(* CODESYS project Storage.project

Project tree, tasks and I/O mapping:
  Storage : CECC-LK, Festo AG & Co. KG, order no. 574418, version 3.5.4.0
    application Application
      libraries: Util, * (System)
      task MainTask (cyclic, interval t#20ms, priority 20) calls Main
      global variables GVL_Storage
      function block FB_BitCode [SFC]: ACT
      function block FB_SeqNTransport_ST [SFC]: ACT
      function block FB_OpMode [FBD]
      program Main [FBD]
    Onboard : CECC 14I/8O, Festo AG & Co. KG, order no. 
      , version 3.4.5.5
        unmapped channels: Onboard Input, Onboard Output
      Digital Inputs
          unmapped channels: Onboard Input
      Digital Outputs
          unmapped channels: Onboard Output
    IO_Link_Master_4_Ports_ : IO-Link Master (4 Ports), Festo AG & Co. KG, order no. 
      , version 3.0.0.3
      BNI_IOL_310_000_K025 : BNI IOL-310-000-K025, Balluff GmbH, version V1.2
          settings:  = 0; ProcessDataID = V_PdT; ProcessDataInLength = 16; ProcessDataOutLength = 16; ProcessDataDescription.bitOffset = 8; ProcessDataDescription.bitLength = 1; ProcessDataDescription.userType = 0; ProcessDataDescription.ChannelType = 1; ProcessDataDescription.bitOffset = 9; ProcessDataDescription.bitLength = 1; ProcessDataDescription.userType = 0; ProcessDataDescription.ChannelType = 1; ProcessDataDescription.bitOffset = 10; ProcessDataDescription.bitLength = 1; ProcessDataDescription.userType = 0; ProcessDataDescription.ChannelType = 1; ProcessDataDescription.bitOffset = 11; ProcessDataDescription.bitLength = 1; ProcessDataDescription.userType = 0; ProcessDataDescription.ChannelType = 1; ProcessDataDescription.bitOffset = 12; ProcessDataDescription.bitLength = 1; ProcessDataDescription.userType = 0; ProcessDataDescription.ChannelType = 1; ProcessDataDescription.bitOffset = 13; ProcessDataDescription.bitLength = 1; ProcessDataDescription.userType = 0; ProcessDataDescription.ChannelType = 1; ProcessDataDescription.bitOffset = 14; ProcessDataDescription.bitLength = 1; ProcessDataDescription.userType = 0; ProcessDataDescription.ChannelType = 1; ProcessDataDescription.bitOffset = 15; ProcessDataDescription.bitLength = 1; ProcessDataDescription.userType = 0; ProcessDataDescription.ChannelType = 1; ProcessDataDescription.bitOffset = 0; ProcessDataDescription.bitLength = 1; ProcessDataDescription.userType = 0; ProcessDataDescription.ChannelType = 1;
            ProcessDataDescription.bitOffset = 1; ProcessDataDescription.bitLength = 1; ProcessDataDescription.userType = 0; ProcessDataDescription.ChannelType = 1; ProcessDataDescription.bitOffset = 2; ProcessDataDescription.bitLength = 1; ProcessDataDescription.userType = 0; ProcessDataDescription.ChannelType = 1; ProcessDataDescription.bitOffset = 3; ProcessDataDescription.bitLength = 1; ProcessDataDescription.userType = 0; ProcessDataDescription.ChannelType = 1; ProcessDataDescription.bitOffset = 4; ProcessDataDescription.bitLength = 1; ProcessDataDescription.userType = 0; ProcessDataDescription.ChannelType = 1; ProcessDataDescription.bitOffset = 5; ProcessDataDescription.bitLength = 1; ProcessDataDescription.userType = 0; ProcessDataDescription.ChannelType = 1; ProcessDataDescription.bitOffset = 6; ProcessDataDescription.bitLength = 1; ProcessDataDescription.userType = 0; ProcessDataDescription.ChannelType = 1; ProcessDataDescription.bitOffset = 7; ProcessDataDescription.bitLength = 1; ProcessDataDescription.userType = 0; ProcessDataDescription.ChannelType = 1; ProcessDataDescription.bitOffset = 8; ProcessDataDescription.bitLength = 1; ProcessDataDescription.userType = 0; ProcessDataDescription.ChannelType = 2; ProcessDataDescription.bitOffset = 9; ProcessDataDescription.bitLength = 1; ProcessDataDescription.userType = 0; ProcessDataDescription.ChannelType = 2; ProcessDataDescription.bitOffset = 10; ProcessDataDescription.bitLength = 1; ProcessDataDescription.userType = 0; ProcessDataDescription.ChannelType = 2;
            ProcessDataDescription.bitOffset = 11; ProcessDataDescription.bitLength = 1; ProcessDataDescription.userType = 0; ProcessDataDescription.ChannelType = 2; ProcessDataDescription.bitOffset = 12; ProcessDataDescription.bitLength = 1; ProcessDataDescription.userType = 0; ProcessDataDescription.ChannelType = 2; ProcessDataDescription.bitOffset = 13; ProcessDataDescription.bitLength = 1; ProcessDataDescription.userType = 0; ProcessDataDescription.ChannelType = 2; ProcessDataDescription.bitOffset = 14; ProcessDataDescription.bitLength = 1; ProcessDataDescription.userType = 0; ProcessDataDescription.ChannelType = 2; ProcessDataDescription.bitOffset = 15; ProcessDataDescription.bitLength = 1; ProcessDataDescription.userType = 0; ProcessDataDescription.ChannelType = 2; ProcessDataDescription.bitOffset = 0; ProcessDataDescription.bitLength = 1; ProcessDataDescription.userType = 0; ProcessDataDescription.ChannelType = 2; ProcessDataDescription.bitOffset = 1; ProcessDataDescription.bitLength = 1; ProcessDataDescription.userType = 0; ProcessDataDescription.ChannelType = 2; ProcessDataDescription.bitOffset = 2; ProcessDataDescription.bitLength = 1; ProcessDataDescription.userType = 0; ProcessDataDescription.ChannelType = 2; ProcessDataDescription.bitOffset = 3; ProcessDataDescription.bitLength = 1; ProcessDataDescription.userType = 0; ProcessDataDescription.ChannelType = 2; ProcessDataDescription.bitOffset = 4; ProcessDataDescription.bitLength = 1; ProcessDataDescription.userType = 0; ProcessDataDescription.ChannelType = 2;
            ProcessDataDescription.bitOffset = 5; ProcessDataDescription.bitLength = 1; ProcessDataDescription.userType = 0; ProcessDataDescription.ChannelType = 2; ProcessDataDescription.bitOffset = 6; ProcessDataDescription.bitLength = 1; ProcessDataDescription.userType = 0; ProcessDataDescription.ChannelType = 2; ProcessDataDescription.bitOffset = 7; ProcessDataDescription.bitLength = 1; ProcessDataDescription.userType = 0; ProcessDataDescription.ChannelType = 2
          unmapped channels: Switchstate Pin 1 (Bit0.0), Switchstate Pin 2 (Bit0.1), Switchstate Pin 3 (Bit0.2), Switchstate Pin 4 (Bit0.3), Switchstate Pin 5 (Bit0.4), Switchstate Pin 6 (Bit0.5), Switchstate Pin 7 (Bit0.6), Switchstate Pin 8 (Bit0.7), Switchstate Pin 9 (Bit1.0), Switchstate Pin 10 (Bit1.1), Switchstate Pin 11 (Bit1.2), Switchstate Pin 12 (Bit1.3), Switchstate Pin 13 (Bit1.4), Switchstate Pin 14 (Bit1.5), Switchstate Pin 15 (Bit1.6), Switchstate Pin 16 (Bit1.7), Switchstate Pin 1 (Bit0.0), Switchstate Pin 2 (Bit0.1), Switchstate Pin 3 (Bit0.2), Switchstate Pin 4 (Bit0.3), Switchstate Pin 5 (Bit0.4), Switchstate Pin 6 (Bit0.5), Switchstate Pin 7 (Bit0.6), Switchstate Pin 8 (Bit0.7), Switchstate Pin 9 (Bit1.0), Switchstate Pin 10 (Bit1.1), Switchstate Pin 11 (Bit1.2), Switchstate Pin 12 (Bit1.3), Switchstate Pin 13 (Bit1.4), Switchstate Pin 14 (Bit1.5), Switchstate Pin 15 (Bit1.6), Switchstate Pin 16 (Bit1.7)
      <Leer>
      <Leer>
      <Leer>
  libraries: Standard, * (System); Util, * (System)
  global variables ToDo
*)

// ToDo
VAR_GLOBAL
END_VAR

// Storage/Application/GVL_Storage
VAR_GLOBAL

//Input			
//Balluf IO-LINK 
xStore_ResetReady	AT	%IX2.0	:BOOL;	//
xStore_Error		AT	%IX2.1	:BOOL;	//
xStore_Busy			AT	%IX2.2	:BOOL;	//
xStore_Full			AT	%IX2.3	:BOOL;	//
xStore_WPAvailable	AT	%IX2.4	:BOOL;	//
xWPnotBlack			AT	%IX2.5	:BOOL;	//
xWPmetallic			AT	%IX2.6	:BOOL;	//
//AT	%IX2.7	:BOOL;	//
	
//CECC-LK Onboard		
SF1 	AT	%IX0.0	:BOOL;	//Taster Start / Start button
SF2 	AT	%IX0.1	:BOOL;	//Taster Stop (Öffner) / Stop Button (normally closed)
SF3 	AT	%IX0.3	:BOOL;	//Taster Richten / Reset button
SF4 	AT	%IX0.2	:BOOL;	//Schlüsselschalter Auto-Manuell / Key Switch auto-manual
XI4		AT	%IX0.4	:BOOL;	//Input from the onboard input pins 
XI5		AT	%IX0.6	:BOOL;	//
XD6 	AT	%IX0.7	:BOOL;	//Folgestation belegt / dwonstream station free			switched address with xd7 for consistency with other stations
XD7		AT	%IX0.5	:BOOL;	//Folgestation belegt / next station free			switched address with xd6 for consistency with other stations
			
//Output	
//Balluf IO-LINK 		//find out how the the xStore_BitCodeBit# is mapped with the IO
xStore_Reference	AT	%QX2.0	:BOOL;	//
xStore_ClearFault	AT	%QX2.1	:BOOL;	//
xStore_Mode			AT	%QX2.2	:BOOL;	// 0 == Store ; 1 == Unstore
xStore_BitCodeBit0	AT	%QX2.3	:BOOL;	//
xStore_BitCodeBit1	AT	%QX2.4	:BOOL;	// 
xStore_BitCodeBit2	AT	%QX2.5	:BOOL;	//
xStore_Strobe		AT	%QX2.6	:BOOL;	//
xStore_Option		AT	%QX2.7	:BOOL;	//
		
//CECC-LK Onboard	
PF1			AT	%QX0.0	:BOOL;	//Leuchtmelder Start / Start indicator light
PF2 		AT	%QX0.1	:BOOL;	//Leuchtmelder Reset / Reset indicator light
PF3 		AT	%QX0.2	:BOOL;	//Leuchte Q1 / Indicator light Q1
PF4			AT	%QX0.3	:BOOL;	//Leuchte Q2 / Indicator light Q2
XD4			AT	%QX0.4	:BOOL;	//Station frei / Station free
indLightGn	AT	%QX0.5	:BOOL;	//Ampel grün / indicator lights green
indLightYe	AT	%QX0.6	:BOOL;	//Ampel gelb / indicator lights yellow
indLightRd 	AT	%QX0.7	:BOOL;	//Apel rot / indicator lights red

// Flags for the Main prg
xStopStoring			:BOOL;
xResetModules			:BOOL;	//Alle Module resetten / Reset all Moduls
xResetReadyModule1		:BOOL;	//Module 1 ist in reset Position / Modul 1 is in reset posisition
xResetReadyModule2		:BOOL;	//Module 2 ist in reset Position / Modul 2 is in reset posisition
xResetReadyModule3		:BOOL;	//Module 3 ist in reset Position / Modul 3 is in reset posisition
xEnAutoMM				:BOOL;	//Automatikmodus aktiv / Automode activated
xDeactivateModules		:BOOL;	//
xProcessBusyMM			:BOOL;	//Station arbeitet / Station is busy
xResetReadyMM			:BOOL;	//Modul SeqTransport ist fertig / Modul SeqTransport is ready
xNextStationFreeMM		:BOOL;	//Nächste Station ist frei / Next Station is free
xReadyModSM				:BOOL;	//Modul ist fertig / Modul is ready
xStartModuleSM			:BOOL;	//Modul starten / Start modul
xInitModules			:BOOL;	//Moduel auf Inischritt setzten / Set moduls to init step
AlwaysTRUE				:BOOL:=TRUE;	//Immer true / Always true
AlwaysFALSE				:BOOL:=FALSE;	//Immer false / Always false
xErrorSignal1			:BOOL;	//Error Signal 1 / Error signal	1
xErrorSignal2			:BOOL;	//Error Signal 2 / Error signal	2
xErrorSignal3			:BOOL;	//Error Signal 3 / Error signal	3

xMKeySwitchOut			:BOOL;
xMStartOut				:BOOL;
xMI4Out					:BOOL;
xMBit0					:BOOL;
xMBit1					:BOOL;
xMBit2					:BOOL;
xMI7Out					:BOOL;
xMPF3					:BOOL;
END_VAR

// Storage/Application/Main
PROGRAM Main//the sequensce of operations 

//for the reference of the variables 
VAR
	FB_OpMode_0				: FB_OpMode; // the initialising code, and for the detection of the colour
	//xMI4Out has something to do with the rising edge from the sensors
	FB_SeqNTransport_ST_0	: FB_SeqNTransport_ST;
	//xMBits are probably for the storage location 
	FB_BitCode_0			: FB_BitCode;
END_VAR

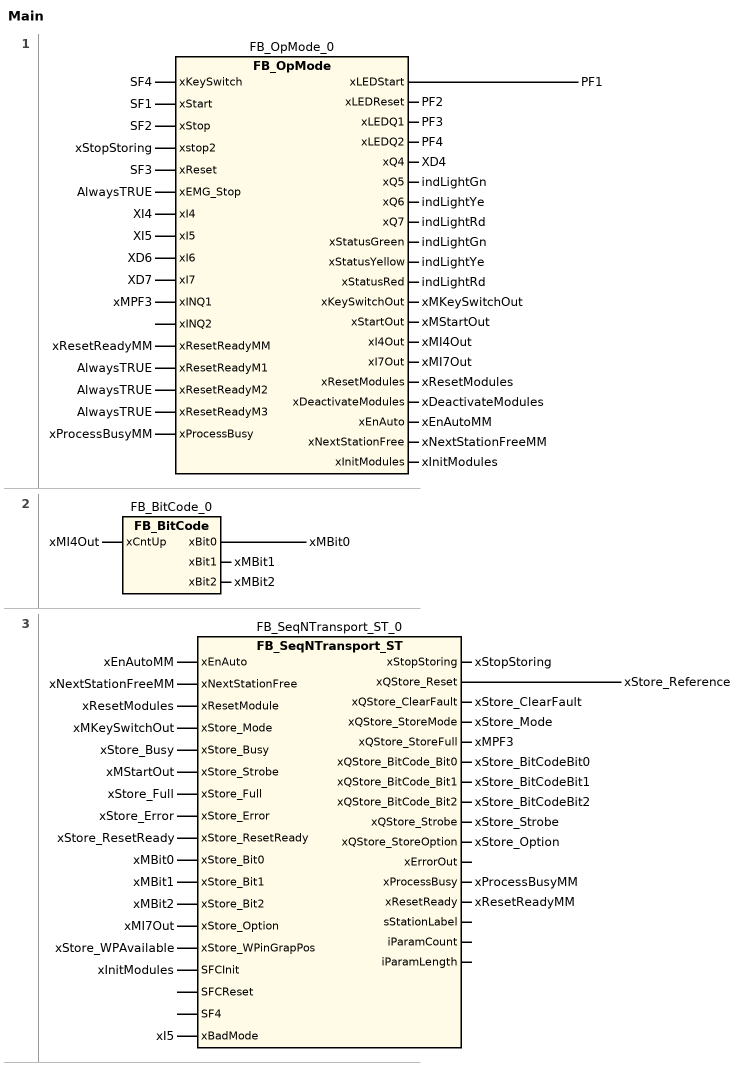
// NETWORK 1
FB_OpMode_0(
    xKeySwitch := SF4,
    xStart := SF1,
    xStop := SF2,
    xstop2 := xStopStoring,
    xReset := SF3,
    xEMG_Stop := AlwaysTRUE,
    xI4 := XI4,
    xI5 := XI5,
    xI6 := XD6,
    xI7 := XD7,
    xINQ1 := xMPF3,
    xResetReadyMM := xResetReadyMM,
    xResetReadyM1 := AlwaysTRUE,
    xResetReadyM2 := AlwaysTRUE,
    xResetReadyM3 := AlwaysTRUE,
    xProcessBusy := xProcessBusyMM,
    xLEDReset => PF2,
    xLEDQ1 => PF3,
    xLEDQ2 => PF4,
    xQ4 => XD4,
    xQ5 => indLightGn,
    xQ6 => indLightYe,
    xQ7 => indLightRd,
    xStatusGreen => indLightGn,
    xStatusYellow => indLightYe,
    xStatusRed => indLightRd,
    xKeySwitchOut => xMKeySwitchOut,
    xStartOut => xMStartOut,
    xI4Out => xMI4Out,
    xI7Out => xMI7Out,
    xResetModules => xResetModules,
    xDeactivateModules => xDeactivateModules,
    xEnAuto => xEnAutoMM,
    xNextStationFree => xNextStationFreeMM,
    xInitModules => xInitModules); // FB_OpMode
PF1 := FB_OpMode_0.xLEDStart;

// NETWORK 2
FB_BitCode_0(xCntUp := xMI4Out, xBit1 => xMBit1, xBit2 => xMBit2); // FB_BitCode
xMBit0 := FB_BitCode_0.xBit0;

// NETWORK 3
FB_SeqNTransport_ST_0(
    xEnAuto := xEnAutoMM,
    xNextStationFree := xNextStationFreeMM,
    xResetModule := xResetModules,
    xStore_Mode := xMKeySwitchOut,
    xStore_Busy := xStore_Busy,
    xStore_Strobe := xMStartOut,
    xStore_Full := xStore_Full,
    xStore_Error := xStore_Error,
    xStore_ResetReady := xStore_ResetReady,
    xStore_Bit0 := xMBit0,
    xStore_Bit1 := xMBit1,
    xStore_Bit2 := xMBit2,
    xStore_Option := xMI7Out,
    xStore_WPinGrapPos := xStore_WPAvailable,
    SFCInit := xInitModules,
    xBadMode := xI5,
    xStopStoring => xStopStoring,
    xQStore_ClearFault => xStore_ClearFault,
    xQStore_StoreMode => xStore_Mode,
    xQStore_StoreFull => xMPF3,
    xQStore_BitCode_Bit0 => xStore_BitCodeBit0,
    xQStore_BitCode_Bit1 => xStore_BitCodeBit1,
    xQStore_BitCode_Bit2 => xStore_BitCodeBit2,
    xQStore_Strobe => xStore_Strobe,
    xQStore_StoreOption => xStore_Option,
    xProcessBusy => xProcessBusyMM,
    xResetReady => xResetReadyMM); // FB_SeqNTransport_ST
xStore_Reference := FB_SeqNTransport_ST_0.xQStore_Reset;

END_PROGRAM

// Storage/Application/FB_OpMode
FUNCTION_BLOCK FB_OpMode
VAR_INPUT
	xKeySwitch 			:BOOL;	//Schlüsselschalter Auto-Manuell / Key Switch auto-manual
	xStart				:BOOL;	//Taster Start / Start button
	xStop				:BOOL;	//Taster Stop (Öffner) / Stop Button (normally closed)
	xstop2				:BOOL;	//Stop when key is switched during operating
	xReset				:BOOL;	//Taster Richten / Reset button
	xEMG_Stop			:BOOL;	//Not Aus Schlagtaster / Emergency Stop
	xI4					:BOOL;	//Bedienfeld Eingang 4 / Panel Input 4
	xI5					:BOOL;	//Bedienfeld Eingang 5 / Panel Input 5
	xI6					:BOOL;	//Folgestation belegt / dwonstream station busy
	xI7					:BOOL;	//Bedienfeld Eingang 7 / Panel Input 7
	xINQ1				:BOOL;	//Eingang Leuchte Q1 / Input Indicator light Q1
	xINQ2				:BOOL;	//Eingang Leuchte Q2 / Input Indicator light Q2
	xResetReadyMM		:BOOL;	//Alle Modul sidn Resetet / Reset ready all Moduls
	xResetReadyM1		:BOOL;	//Modul 1 ist Resetet / Reset ready Modul 1
	xResetReadyM2		:BOOL;	//Modul 2 ist Resetet / Reset ready Modul 2
	xResetReadyM3		:BOOL;	//Modul 3 ist Resetet / Reset ready Modul 3
	xProcessBusy		:BOOL;	//Station belegt / Station is busy
END_VAR
VAR_OUTPUT
	xLEDStart			:BOOL;	//Leuchtmelder Start / Start indicator light
	xLEDReset			:BOOL;	//Leuchtmelder Reset / Reset indicator light
	xLEDQ1				:BOOL;	//Leuchte Q1 / Indicator light Q1
	xLEDQ2				:BOOL;	//Leuchte Q2 / Indicator light Q2
	xQ4					:BOOL;	//Station frei / Station free / Bedienfeld Ausgang 4 / Panel Output 4
	xQ5					:BOOL;	//Bedienfeld Ausgang 5 / Panel Output 5
	xQ6					:BOOL;	//Bedienfeld Ausgang 6 / Panel Output 6
	xQ7					:BOOL;	//Bedienfeld Ausgang 7 / Panel Output 7
	xStatusGreen		:BOOL;	//Ampel grün / indicator lights green
	xStatusYellow		:BOOL;	//Ampel gelb / indicator lights yellow
	xStatusRed			:BOOL;	//Apel rot / indicator lights red
	xKeySwitchOut		:BOOL;
	xStartOut			:BOOL;
	xI4Out				:BOOL;
	xI7Out				:BOOL;
	xResetModules		:BOOL;	//Module reseten / Reset Moduls
	xDeactivateModules	:BOOL;	//Module deaktivieren / Deactivate Moduls
	xEnAuto				:BOOL;	//Automatikbetrieb / Automatic mode
	xNextStationFree	:BOOL;	//Folgestation frei / Next Station is free
	xInitModules		:BOOL;	//Moduls auf Initial Schritt setzten / Set Moduls Initial step
END_VAR
VAR
	test				:BOOL;
	FirstScan			:BOOL := 1;	//Always true
	
	RESETALL			:BOOL;	
	xBlockPositive		:BOOL;	
	xBlockNegative		:BOOL;	
	xResetReadyModules	:BOOL;	
	xclock_Green		:BOOL;	
	xclock_Yellow		:BOOL;	
	N_Trig_ResetModules	:BOOL;	
	xLED				:SR;
	MANUAL				:SR;	
	AutoEN				:SR;	
	RESET				:SR;
	MANUALIND			:SR;
	INITIAL				:SR;	
	BLINK_1Hz			:Blink;
	F_TRIG_ResetERR		:F_TRIG;	
	VarTimeCur			:TIME;
	RESETSAVE			:SR;
	T_ResetTimer: TON;
	T_StopTimer: TON;
	BLINK_Q1: Blink;
	TOF_Q1: TOF;
	TP_Q1: TP;
		Key_Switch: R_TRIG;
	Key_Switch2: F_TRIG;
	xKeyswitch_stop: BOOL;
END_VAR
VAR // added by the converter: edge detectors and wires of the graphical bodies
    _w1 : BOOL;
END_VAR

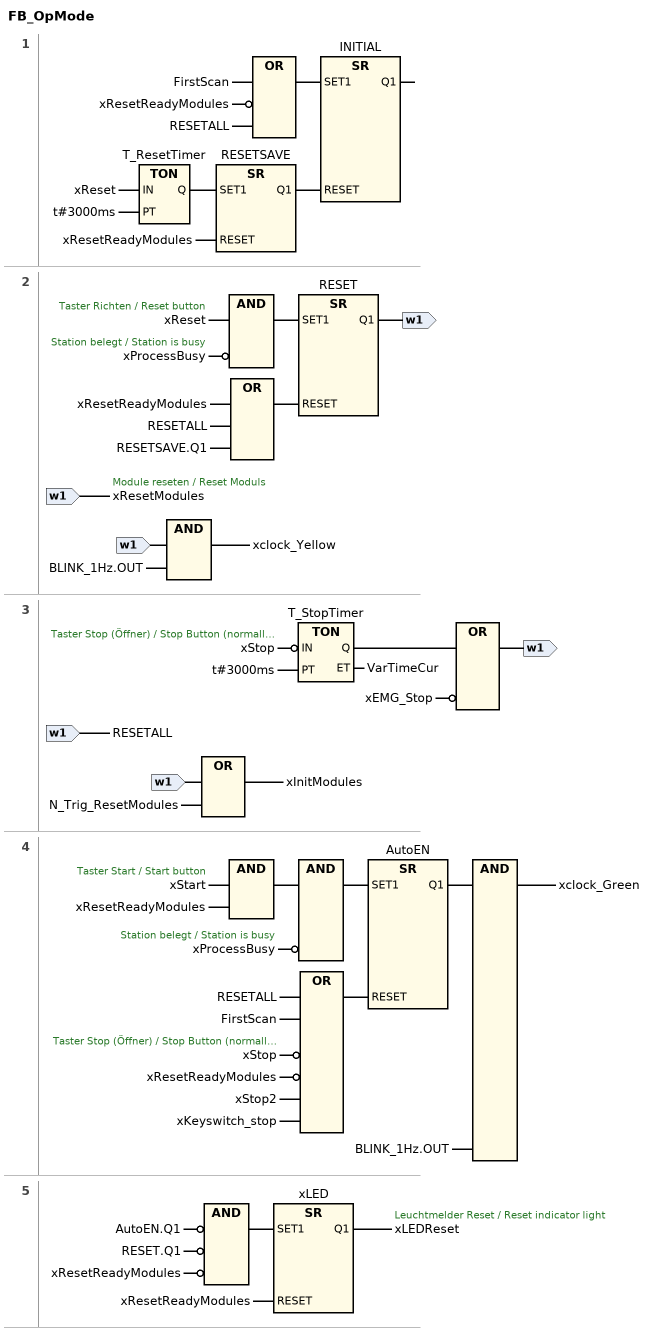
// NETWORK 1
T_ResetTimer(IN := xReset, PT := t#3000ms); // TON
RESETSAVE(SET1 := T_ResetTimer.Q, RESET := xResetReadyModules); // SR
INITIAL(SET1 := FirstScan OR NOT xResetReadyModules OR RESETALL, RESET := RESETSAVE.Q1); // SR

// NETWORK 2
//   xReset: Taster Richten / Reset button
//   xProcessBusy: Station belegt / Station is busy
//   xResetModules: Module reseten / Reset Moduls
RESET(SET1 := xReset AND NOT xProcessBusy, RESET := xResetReadyModules OR RESETALL OR RESETSAVE.Q1); // SR
xResetModules := RESET.Q1;
xclock_Yellow := RESET.Q1 AND BLINK_1Hz.OUT;

// NETWORK 3
//   xStop: Taster Stop (Öffner) / Stop Button (normally closed)
T_StopTimer(IN := NOT xStop, PT := t#3000ms, ET => VarTimeCur); // TON
_w1 := T_StopTimer.Q OR NOT xEMG_Stop;
RESETALL := _w1;
xInitModules := _w1 OR N_Trig_ResetModules;

// NETWORK 4
//   xStart: Taster Start / Start button
//   xProcessBusy: Station belegt / Station is busy
//   xStop: Taster Stop (Öffner) / Stop Button (normally closed)
AutoEN(SET1 := (xStart AND xResetReadyModules) AND NOT xProcessBusy, RESET := RESETALL OR FirstScan OR NOT xStop OR NOT xResetReadyModules OR xStop2 OR xKeyswitch_stop); // SR
xclock_Green := AutoEN.Q1 AND BLINK_1Hz.OUT;

// NETWORK 5
//   xLEDReset: Leuchtmelder Reset / Reset indicator light
xLED(SET1 := NOT AutoEN.Q1 AND NOT RESET.Q1 AND NOT xResetReadyModules, RESET := xResetReadyModules); // SR
xLEDReset := xLED.Q1;

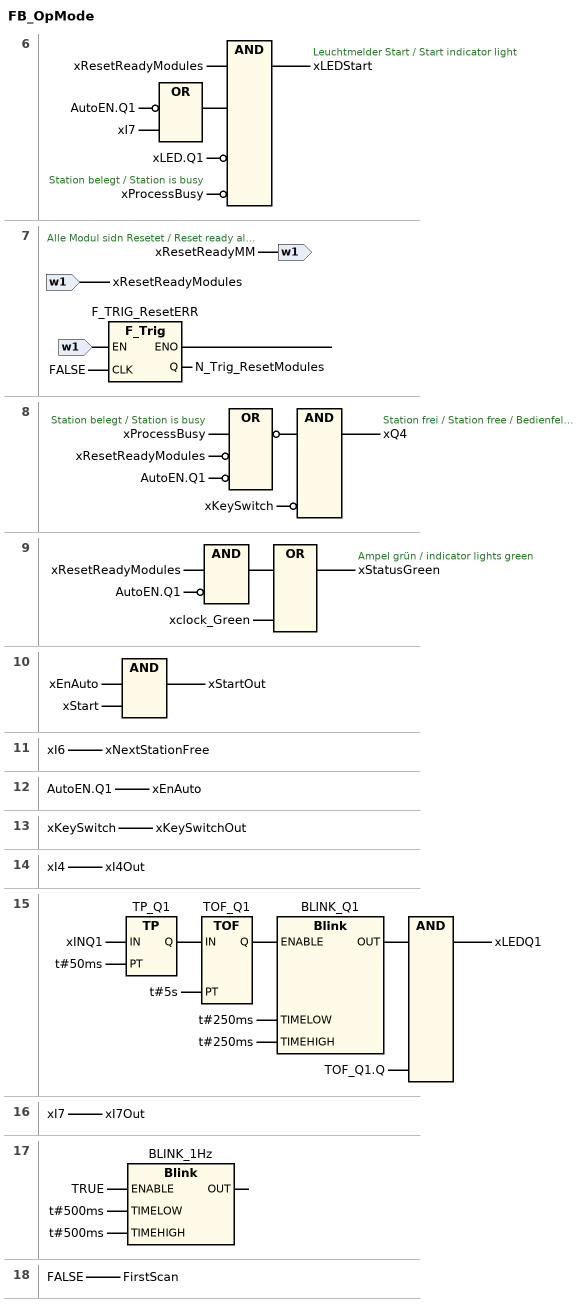
// NETWORK 6
//   xProcessBusy: Station belegt / Station is busy
//   xLEDStart: Leuchtmelder Start / Start indicator light
xLEDStart := xResetReadyModules AND (NOT AutoEN.Q1 OR xI7) AND NOT xLED.Q1 AND NOT xProcessBusy;

// NETWORK 7
//   xResetReadyMM: Alle Modul sidn Resetet / Reset ready all Moduls
xResetReadyModules := xResetReadyMM;
IF xResetReadyMM THEN
    F_TRIG_ResetERR(CLK := FALSE, Q => N_Trig_ResetModules); // F_Trig
END_IF

// NETWORK 8
//   xProcessBusy: Station belegt / Station is busy
//   xQ4: Station frei / Station free / Bedienfeld Ausgang 4 / Panel Output 4
xQ4 := NOT (xProcessBusy OR NOT xResetReadyModules OR NOT AutoEN.Q1) AND NOT xKeySwitch;

// NETWORK 9
//   xStatusGreen: Ampel grün / indicator lights green
xStatusGreen := xResetReadyModules AND NOT AutoEN.Q1 OR xclock_Green;

// NETWORK 10
xStartOut := xEnAuto AND xStart;

// NETWORK 11
xNextStationFree := xI6;

// NETWORK 12
xEnAuto := AutoEN.Q1;

// NETWORK 13
xKeySwitchOut := xKeySwitch;

// NETWORK 14
xI4Out := xI4;

// NETWORK 15
TP_Q1(IN := xINQ1, PT := t#50ms); // TP
TOF_Q1(IN := TP_Q1.Q, PT := t#5s); // TOF
BLINK_Q1(ENABLE := TOF_Q1.Q, TIMELOW := t#250ms, TIMEHIGH := t#250ms); // Blink
xLEDQ1 := BLINK_Q1.OUT AND TOF_Q1.Q;

// NETWORK 16
xI7Out := xI7;

// NETWORK 17
BLINK_1Hz(ENABLE := TRUE, TIMELOW := t#500ms, TIMEHIGH := t#500ms); // Blink

// NETWORK 18
FirstScan := FALSE;

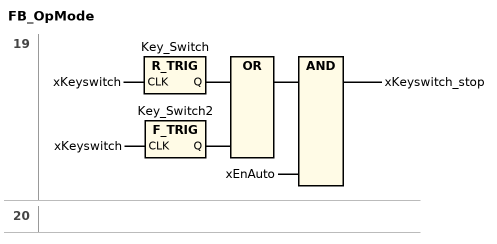
// NETWORK 19
Key_Switch(CLK := xKeyswitch); // R_TRIG
Key_Switch2(CLK := xKeyswitch); // F_TRIG
xKeyswitch_stop := (Key_Switch.Q OR Key_Switch2.Q) AND xEnAuto;

// NETWORK 20

END_FUNCTION_BLOCK

// Storage/Application/FB_BitCode
FUNCTION_BLOCK FB_BitCode // this code gives the output as a bit depending on the colour of the workpiece from the rising edge detector
VAR_INPUT
	xCntUp			:BOOL;
END_VAR
VAR_OUTPUT
	xBit0			:BOOL;
	xBit1			:BOOL;
	xBit2			:BOOL;
	
END_VAR
VAR
	R_TRIG_CntUp	:R_Trig;
END_VAR

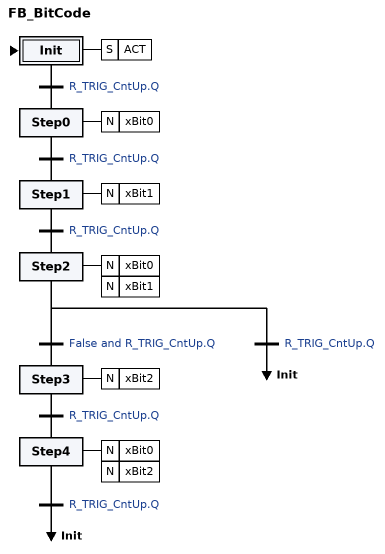
INITIAL_STEP Init:
    ACT(S);
END_STEP
TRANSITION FROM Init TO Step0
    := R_TRIG_CntUp.Q;
END_TRANSITION
STEP Step0:
    xBit0(N);
END_STEP
TRANSITION FROM Step0 TO Step1
    := R_TRIG_CntUp.Q;
END_TRANSITION
STEP Step1:
    xBit1(N);
END_STEP
TRANSITION FROM Step1 TO Step2
    := R_TRIG_CntUp.Q;
END_TRANSITION
STEP Step2:
    xBit0(N);
    xBit1(N);
END_STEP
TRANSITION FROM Step2 TO Step3
    := False and R_TRIG_CntUp.Q;
END_TRANSITION
TRANSITION FROM Step2 TO Init
    := R_TRIG_CntUp.Q;
END_TRANSITION
STEP Step3:
    xBit2(N);
END_STEP
TRANSITION FROM Step3 TO Step4
    := R_TRIG_CntUp.Q;
END_TRANSITION
STEP Step4:
    xBit0(N);
    xBit2(N);
END_STEP
TRANSITION FROM Step4 TO Init
    := R_TRIG_CntUp.Q;
END_TRANSITION

ACTION ACT:
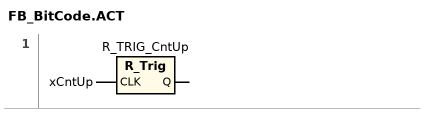
// NETWORK 1
R_TRIG_CntUp(CLK := xCntUp); // R_Trig
END_ACTION

END_FUNCTION_BLOCK

// Storage/Application/FB_SeqNTransport_ST
FUNCTION_BLOCK FB_SeqNTransport_ST
VAR_INPUT
	xEnAuto					:BOOL;	//Automatikbetrieb / Automatic mode
	xNextStationFree		:BOOL;	//Folgestation Frei / Next Station is Free
	xResetModule			:BOOL;	//Module sind resetet / Moduls in reset position
	xStore_Mode				:BOOL;
	xStore_Busy				:BOOL;
	xStore_Strobe			:BOOL;
	xStore_Full				:BOOL;
	xStore_Error			:BOOL;
	xStore_ResetReady		:BOOL;
	xStore_Bit0				:BOOL;
	xStore_Bit1				:BOOL;
	xStore_Bit2				:BOOL;
k
END_VAR
VAR_OUTPUT
xStopStoring 					:BOOL;	
xQStore_Reset			:BOOL;
	xQStore_ClearFault		:BOOL;
	xQStore_StoreMode		:BOOL;
	xQStore_StoreFull		:BOOL;
	xQStore_BitCode_Bit0	:BOOL;
	xQStore_BitCode_Bit1	:BOOL;
	xQStore_BitCode_Bit2	:BOOL;
	xQStore_Strobe			:BOOL;
	xQStore_StoreOption		:BOOL;
	xErrorOut				:BOOL;	//Fehler Ausgang / Error Output
	xProcessBusy			:BOOL;	//Station Belegt / Station busy	
	xResetReady				:BOOL;	//Prg. Transport Reset ist fertig / Reset ready Prg. Trpansport
	sStationLabel			:STRING;//Stations Name / Station Label
	iParamCount				:INT;	//Parameter Anzahl / Paramerter count
	iParamLength			:INT;	//Parameter Länge / Parameter length
END_VAR					
VAR
	xPulseStrobe			:BOOL;
	xTempQ1					:BOOL;
	xTempQ1_2				:BOOL;
	xClock_2_5Hz			:BOOL;
	R_TRIG_Strobe			:R_Trig;
	sStationName			:STRING:='ST';	//Stations Name / Station Label
	IEC_Timer_0_BlockStrobe	:TON;
	IEC_Timer_0_PulseStrobe	:TP;
	BLINK_2_5Hz: Blink;
	ShortCycleRunning:BOOL;
	LongCycleRunning:BOOL;
END_VAR

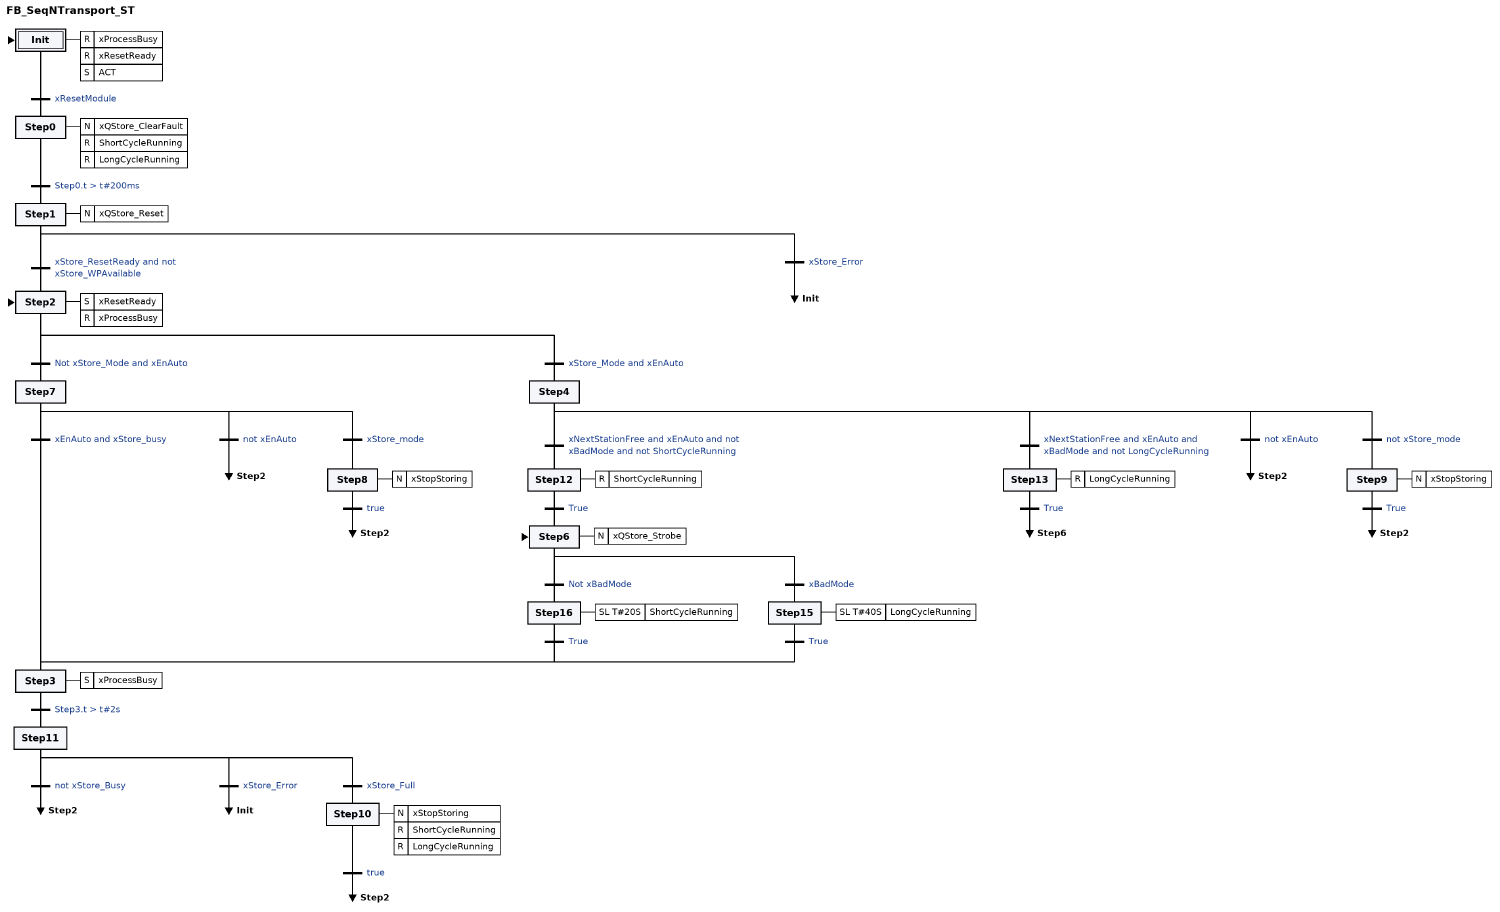
INITIAL_STEP Init:
    xProcessBusy(R);
    xResetReady(R);
    ACT(S);
END_STEP
TRANSITION FROM Init TO Step0
    := xResetModule;
END_TRANSITION
STEP Step0:
    xQStore_ClearFault(N);
    ShortCycleRunning(R);
    LongCycleRunning(R);
END_STEP
TRANSITION FROM Step0 TO Step1
    := Step0.t > t#200ms;
END_TRANSITION
STEP Step1:
    xQStore_Reset(N);
END_STEP
TRANSITION FROM Step1 TO Step2
    := xStore_ResetReady and not xStore_WPAvailable;
END_TRANSITION
TRANSITION FROM Step1 TO Init
    := xStore_Error;
END_TRANSITION
STEP Step2:
    xResetReady(S);
    xProcessBusy(R);
END_STEP
TRANSITION FROM Step2 TO Step7
    := Not xStore_Mode and xEnAuto;
END_TRANSITION
STEP Step7:
END_STEP
TRANSITION FROM Step7 TO Step3
    := xEnAuto and xStore_busy;
END_TRANSITION
TRANSITION FROM Step7 TO Step2
    := not xEnAuto;
END_TRANSITION
TRANSITION FROM Step7 TO Step8
    := xStore_mode;
END_TRANSITION
STEP Step8:
    xStopStoring(N);
END_STEP
TRANSITION FROM Step8 TO Step2
    := true;
END_TRANSITION
TRANSITION FROM Step2 TO Step4
    := xStore_Mode and xEnAuto;
END_TRANSITION
STEP Step4:
END_STEP
TRANSITION FROM Step4 TO Step12
    := xNextStationFree and xEnAuto and not xBadMode and not ShortCycleRunning;
END_TRANSITION
TRANSITION FROM Step4 TO Step13
    := xNextStationFree and xEnAuto and xBadMode and not LongCycleRunning;
END_TRANSITION
STEP Step13:
    LongCycleRunning(R);
END_STEP
TRANSITION FROM Step13 TO Step6
    := True;
END_TRANSITION
STEP Step12:
    ShortCycleRunning(R);
END_STEP
TRANSITION FROM Step12 TO Step6
    := True;
END_TRANSITION
TRANSITION FROM Step4 TO Step2
    := not xEnAuto;
END_TRANSITION
TRANSITION FROM Step4 TO Step9
    := not xStore_mode;
END_TRANSITION
STEP Step9:
    xStopStoring(N);
END_STEP
TRANSITION FROM Step9 TO Step2
    := True;
END_TRANSITION
STEP Step6:
    xQStore_Strobe(N);
END_STEP
TRANSITION FROM Step6 TO Step16
    := Not xBadMode;
END_TRANSITION
STEP Step16:
    ShortCycleRunning(SL, T#20S);
END_STEP
TRANSITION FROM Step16 TO Step3
    := True;
END_TRANSITION
TRANSITION FROM Step6 TO Step15
    := xBadMode;
END_TRANSITION
STEP Step15:
    LongCycleRunning(SL, T#40S);
END_STEP
TRANSITION FROM Step15 TO Step3
    := True;
END_TRANSITION
STEP Step3:
    xProcessBusy(S);
END_STEP
TRANSITION FROM Step3 TO Step11
    := Step3.t > t#2s;
END_TRANSITION
STEP Step11:
END_STEP
TRANSITION FROM Step11 TO Step2
    := not xStore_Busy;
END_TRANSITION
TRANSITION FROM Step11 TO Init
    := xStore_Error;
END_TRANSITION
TRANSITION FROM Step11 TO Step10
    := xStore_Full;
END_TRANSITION
STEP Step10:
    xStopStoring(N);
    ShortCycleRunning(R);
    LongCycleRunning(R);
END_STEP
TRANSITION FROM Step10 TO Step2
    := true;
END_TRANSITION

ACTION ACT:
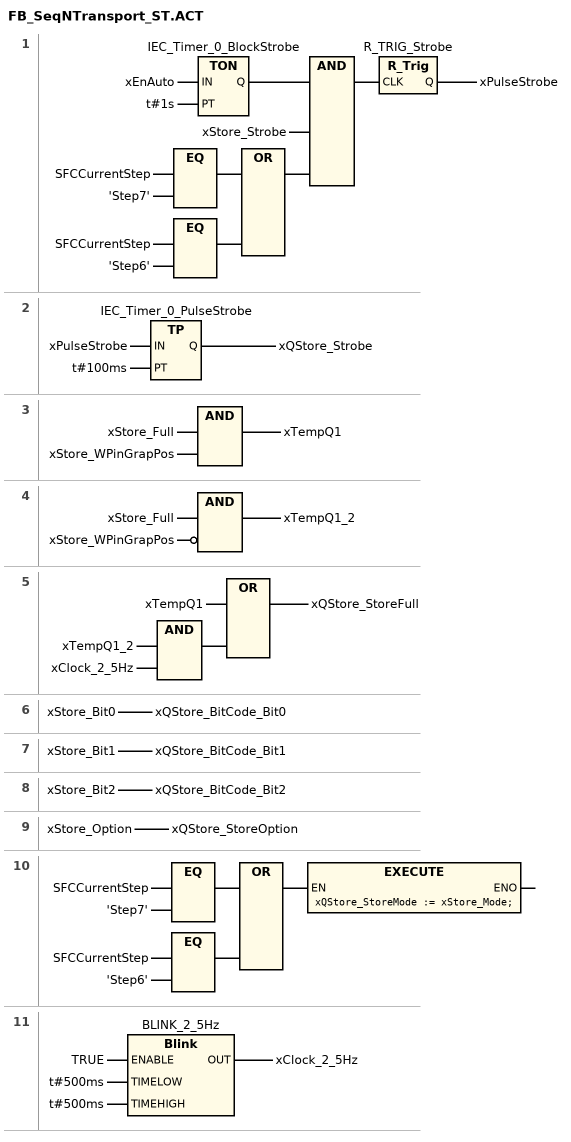
// NETWORK 1
IEC_Timer_0_BlockStrobe(IN := xEnAuto, PT := t#1s); // TON
R_TRIG_Strobe(CLK := IEC_Timer_0_BlockStrobe.Q AND xStore_Strobe AND (SFCCurrentStep = 'Step7' OR SFCCurrentStep = 'Step6')); // R_Trig
xPulseStrobe := R_TRIG_Strobe.Q;

// NETWORK 2
IEC_Timer_0_PulseStrobe(IN := xPulseStrobe, PT := t#100ms); // TP
xQStore_Strobe := IEC_Timer_0_PulseStrobe.Q;

// NETWORK 3
xTempQ1 := xStore_Full AND xStore_WPinGrapPos;

// NETWORK 4
xTempQ1_2 := xStore_Full AND NOT xStore_WPinGrapPos;

// NETWORK 5
xQStore_StoreFull := xTempQ1 OR xTempQ1_2 AND xClock_2_5Hz;

// NETWORK 6
xQStore_BitCode_Bit0 := xStore_Bit0;

// NETWORK 7
xQStore_BitCode_Bit1 := xStore_Bit1;

// NETWORK 8
xQStore_BitCode_Bit2 := xStore_Bit2;

// NETWORK 9
xQStore_StoreOption := xStore_Option;

// NETWORK 10
IF SFCCurrentStep = 'Step7' OR SFCCurrentStep = 'Step6' THEN xQStore_StoreMode := xStore_Mode; END_IF

// NETWORK 11
BLINK_2_5Hz(ENABLE := TRUE, TIMELOW := t#500ms, TIMEHIGH := t#500ms); // Blink
xClock_2_5Hz := BLINK_2_5Hz.OUT;
END_ACTION

END_FUNCTION_BLOCK
